FUNCTION_BLOCK FBiFilter
VAR_INPUT
	bExecute : BOOL;
	ptInputValue : POINTER TO INT;
	ptFilterArray : POINTER TO ARRAY [0..0] OF INT;
	iBufferSize: INT;
END_VAR
VAR_OUTPUT
	bRingbufferFilled : BOOL;
	iFilterOutput : INT;
	fFilterOutput : LREAL;
END_VAR
VAR
	FilterSum : LREAL;
	iPtBufferPointer : INT;
	iValueCount : INT;
END_VAR

IF bExecute THEN
	FilterSum := FilterSum - ptFilterArray^[iPtBufferPointer];
	ptFilterArray^[iPtBufferPointer] := ptInputValue^;
	FilterSum := FilterSum + ptInputValue^;
	iPtBufferPointer := iGetNextBufferPointer(iBufferSize, iPtBufferPointer);
	iFilterOutput := LREAL_TO_INT(FilterSum / INT_TO_LREAL(iBufferSize));
	fFilterOutput := FilterSum / INT_TO_LREAL(iBufferSize);
	IF iValueCount >= iBufferSize THEN
		bRingbufferFilled := 1;
	ELSE
		iValueCount := iValueCount + 1;
	END_IF;
ELSE
	iValueCount := 0;
	bRingbufferFilled := 0;
END_IF;

END_FUNCTION_BLOCK

(* stored: Version 1.1.0.1, ProductVersion 3.1.4024.13
   POU FBiFilter: Id {fb4bdf37-50ff-49d7-91eb-c010553d18d0}, SpecialFunc None *)
